FUNCTION_BLOCK QX_Data_Preparation (* Basic FB with empty ECC *)
  (* Standard: 61499-2 *)
  (* Version 1.0, 2023-03-16, AK125171 *)
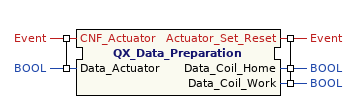
  EVENT_INPUT
    CNF_Actuator WITH Data_Actuator;
  END_EVENT
  EVENT_OUTPUT
    Actuator_Set_Reset WITH Data_Coil_Home, Data_Coil_Work;
  END_EVENT
  VAR_INPUT
    Data_Actuator : BOOL;
  END_VAR
  VAR_OUTPUT
    Data_Coil_Home : BOOL;
    Data_Coil_Work : BOOL;
  END_VAR
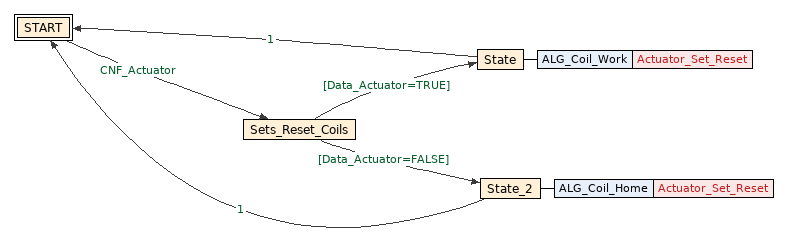
  EC_STATES
    START; (* Initial State *)
    State : ALG_Coil_Work -> Actuator_Set_Reset;
    Sets_Reset_Coils;
    State_2 : ALG_Coil_Home -> Actuator_Set_Reset;
  END_STATES
  EC_TRANSITIONS
    START TO Sets_Reset_Coils := CNF_Actuator;
    Sets_Reset_Coils TO State := [Data_Actuator=TRUE];
    Sets_Reset_Coils TO State_2 := [Data_Actuator=FALSE];
    State TO START := 1;
    State_2 TO START := 1;
  END_TRANSITIONS
  ALGORITHM ALG_Coil_Work IN ST:
Data_Coil_Work:=TRUE;
Data_Coil_Home:=FALSE;
  END_ALGORITHM
  ALGORITHM ALG_Coil_Home IN ST:
Data_Coil_Home:=TRUE;
Data_Coil_Work:=FALSE;
  END_ALGORITHM
END_FUNCTION_BLOCK
